TYPE ST_ClusteringParams :
STRUCT
	nKmppK					:	UDINT 	:=	2;
	bKmppDoublePrecision	:	BOOL 	:=	FALSE;	// optional Exp parameter
	nKmppMaxIterations		:	UDINT	:=	10;		// optional Exp parameter
	fKmppEpsilon			:	LREAL	:=	0.001;	// optional Exp parameter
	nLbgMaxClusters			:	UDINT	:=	5;
	fLbgMaxClusterRadius	:	LREAL	:=	0.6;
	bLbgSingleSplitSteps	:	BOOL	:=	TRUE;
	bLbgDoublePrecision		:	BOOL	:=	FALSE;	// optional Exp parameter
	nLbgMaxIterations		:	UDINT	:=	10;		// optional Exp parameter
	fLbgEpsilon				:	LREAL	:=	0.001;	// optional Exp parameter
	fStaRho	                :	LREAL	:=	0.78;
	nStaNu	                :	UDINT	:=	3;		// optional Exp parameter
	bStaDoublePrecision		:	BOOL	:=	FALSE;	// optional Exp parameter
	fStaBetaSbm				:	LREAL	:=	0.0;	// optional Exp parameter
	nStaPhi					:	UDINT	:=	1;		// optional Exp parameter
	nStaTau					:	UDINT	:=	100;	// optional Exp parameter
END_STRUCT
END_TYPE

(* stored: Version 1.1.0.1, ProductVersion 3.1.4024.12
   DUT ST_ClusteringParams: Id {c46ba47b-cd3b-4f47-b69e-0730d1f6595b} *)
